FUNCTION_BLOCK FB_PartMonitoring_fixt1
VAR_INPUT
END_VAR
VAR_OUTPUT
	
	qRawPart1:BOOL;
	qRawPart2:BOOL;
	qRawPart3:BOOL;
	qRawPart4:BOOL;
	qAllPartPresent:BOOL;
	
END_VAR
VAR
END_VAR

qRawPart1:= (
             fixt2.I.i_PART_CONTROL_B1 AND fixt2.I.i_PART_CONTROL_B2 AND fixt2.I.i_PART_CONTROL_B3 AND fixt2.I.i_PART_CONTROL_B4
			 AND fixt2.I.i_PART_CONTROL_B5 AND fixt2.I.i_PART_CONTROL_B6 AND fixt2.I.i_PART_CONTROL_B7
			 );
qRawPart2:= (
             fixt2.I.i_PART_CONTROL_B15 AND fixt2.I.i_PART_CONTROL_B16 AND fixt2.I.i_PART_CONTROL_B17 AND fixt2.I.i_PART_CONTROL_B18
			 AND fixt2.I.i_PART_CONTROL_B19 AND fixt2.I.i_PART_CONTROL_B20 AND fixt2.I.i_PART_CONTROL_B21
			 );
qRawPart3:= (
             fixt2.I.i_PART_CONTROL_B8 AND fixt2.I.i_PART_CONTROL_B9 AND fixt2.I.i_PART_CONTROL_B10 AND fixt2.I.i_PART_CONTROL_B11
			 AND fixt2.I.i_PART_CONTROL_B12 AND fixt2.I.i_PART_CONTROL_B13 AND fixt2.I.i_PART_CONTROL_B14
			 );
qRawPart4:= (
             fixt2.I.i_PART_CONTROL_B22 AND fixt2.I.i_PART_CONTROL_B23 AND fixt2.I.i_PART_CONTROL_B24 AND fixt2.I.i_PART_CONTROL_B25
			 AND fixt2.I.i_PART_CONTROL_B26 AND fixt2.I.i_PART_CONTROL_B27 AND fixt2.I.i_PART_CONTROL_B28
			 );			 
			 
qAllPartPresent:= (
             fixt2.I.i_PART_CONTROL_B22 AND fixt2.I.i_PART_CONTROL_B23 AND fixt2.I.i_PART_CONTROL_B24 AND fixt2.I.i_PART_CONTROL_B25
			 AND fixt2.I.i_PART_CONTROL_B26 AND fixt2.I.i_PART_CONTROL_B27 AND fixt2.I.i_PART_CONTROL_B28
			 AND fixt2.I.i_PART_CONTROL_B1 AND fixt2.I.i_PART_CONTROL_B2 AND fixt2.I.i_PART_CONTROL_B3 AND fixt2.I.i_PART_CONTROL_B4
			 AND fixt2.I.i_PART_CONTROL_B5 AND fixt2.I.i_PART_CONTROL_B6 AND fixt2.I.i_PART_CONTROL_B7
			 AND fixt2.I.i_PART_CONTROL_B15 AND fixt2.I.i_PART_CONTROL_B16 AND fixt2.I.i_PART_CONTROL_B17 AND fixt2.I.i_PART_CONTROL_B18
			 AND fixt2.I.i_PART_CONTROL_B19 AND fixt2.I.i_PART_CONTROL_B20 AND fixt2.I.i_PART_CONTROL_B21
             AND fixt2.I.i_PART_CONTROL_B8 AND fixt2.I.i_PART_CONTROL_B9 AND fixt2.I.i_PART_CONTROL_B10 AND fixt2.I.i_PART_CONTROL_B11
			 AND fixt2.I.i_PART_CONTROL_B12 AND fixt2.I.i_PART_CONTROL_B13 AND fixt2.I.i_PART_CONTROL_B14 
			 );

END_FUNCTION_BLOCK

(* stored: Version 1.1.0.1, ProductVersion 3.1.4024.16
   POU FB_PartMonitoring_Fixt1: Id {80a4fce0-0737-45b1-906a-8f24ee512c45}, SpecialFunc None *)
